PROGRAM MAIN_1
VAR
	bTest: BOOL;
	Ax1_FB_HomeBeforeMoveAX8000: FB_HomeBeforeMoveAX8000;
END_VAR
VAR PERSISTENT
	nTest : INT;
END_VAR

//Axis01
Axis01_Alarm();
Axis01_Auto();
Axis01_Interlock();
Axis01_Manual();
Axis01_Product_Position();
Axis01_Status();
//Axis02
Axis02_Alarm();
Axis02_Auto();
Axis02_Interlock();
Axis02_Manual();
Axis02_Status();
//Axis03
Axis03_Alarm();
Axis03_Auto();
Axis03_Interlock();
Axis03_Manual();
Axis03_Status();
//Axis04
Axis04_Alarm();
Axis04_Auto();
Axis04_Interlock();
Axis04_Manual();
Axis04_Status();
//Axis05
Axis05_Alarm();
Axis05_Auto();
Axis05_Interlock();
Axis05_Manual();
Axis05_Status();


Alarm();
Axis01_Command();
Axis02_X();
Axis03_Y();
Axis04_Z();
Axis05_Rotation();
Conveyor();
HMI();
System();
Vision();
Main_Step();
Calibration();
HOME_MOVE();

END_PROGRAM

(* stored: Version 1.1.0.1, ProductVersion 3.1.4024.15
   POU MAIN_1: Id {0143168f-bc29-4df3-a416-c4765796282e}, SpecialFunc None *)
